Staubli VAL3: ActiviteEleve.pjx

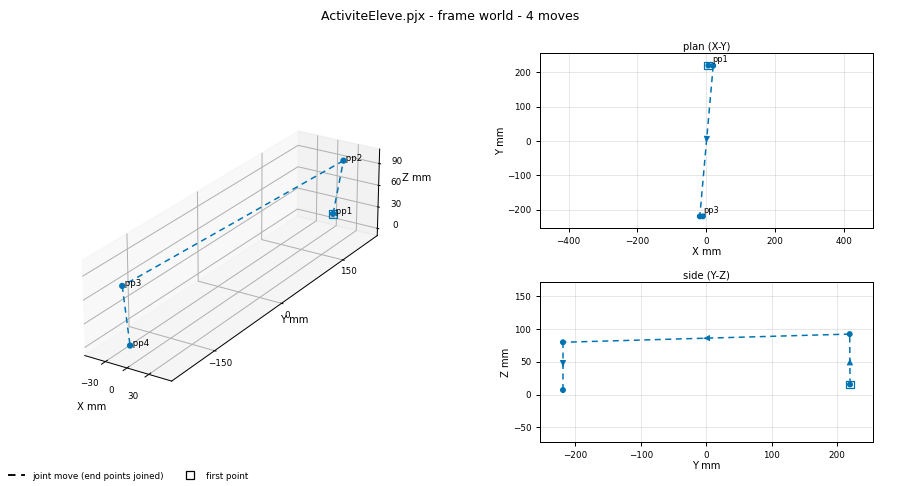
[picture p0: tool path of ActiviteEleve.pjx in frame world, 4 of 6 moves have a stored position in this frame; points joined in program order, loops and branches not executed]
--- ActiviteEleve.pjx ---
Parameters version=s7.11 stackSize=5000 millimeterUnit=true
Program file=check.pgx
Program file=comunication.pgx
Program file=coucou.pgx
Program file=jump.pgx
Program file=PickAndPlace.pgx
Program file=start.pgx
Program file=stop.pgx
Data file=ActiviteEleve.dtx
Library alias=io path=Disk://io/io.pjx

--- ActiviteEleve.dtx ---
pointRs pp1 = {x=6.500000, y=219.500000, z=15.500000, rx=-180, ry=-5.500000e-15, rz=-55.000000, fatherId=world[0]}
pointRs pp2 = {x=20.500000, y=219.000000, z=92.500000, rx=-180, ry=-5.500000e-15, rz=-55.000000, fatherId=world[0]}
pointRs pp3 = {x=-18.500000, y=-219.000000, z=80.000000, rx=180, ry=5.500000e-15, rz=125.500000, fatherId=world[0]}
pointRs pp4 = {x=-9.500000, y=-219.000000, z=7.000000, rx=180, ry=5.500000e-15, rz=123.000000, fatherId=world[0]}

--- start.pgx ---
program start()
begin
  // clean the screen
  userPage()
  cls()
  // create the 2 task
  taskCreate "comunication",10,comunication()
  delay(0.1)
  taskCreate "check",10,check()
end

--- check.pgx ---
program check()
begin
  while taskStatus("comunication")!=-1
    if taskStatus("comunication")>1
      // try to clear the buffer and resume
      clearBuffer(io:tcp_client)
      taskKill("comunication")
      wait(taskStatus("comunication")==-1)
      // create the task again from the beginning
      taskCreate "comunication",10,comunication()
    endIf
    delay(0)
  endWhile
end

--- comunication.pgx ---
program comunication()
  local string sChoixMode
  local string sClient
begin
  // clear the buffer
  clearBuffer(io:tcp_server)
  sClient="Connexion reussie"
  io:tcp_server=sClient

  putln("Un client est connecté")

  while(isKeyPressed(255)==false)
    // write
    sClient="Attente de consigne"
    io:tcp_server=sClient

    // read
    sChoixMode=io:tcp_server
    putln("Mode choisi: "+sChoixMode)

    switch sChoixMode
      //Mode coucou
      case "1"
        //on supprime les tâches en cours
        if taskStatus("jump") != -1
          taskKill("jump")
        endIf
        if taskStatus("pick&place") != -1
          taskKill("pick&place")
        endIf

        delay(0.5)

        putln("Lancement du mode coucou")
        taskCreate "coucou", 10, coucou()
      break
      //Mode jump
      case "2"
        if taskStatus("coucou") != -1
          taskKill("coucou")
        endIf
        if taskStatus("pick&place") != -1
          taskKill("pick&place")
        endIf

        delay(0.5)

        putln("Lancement du mode jump")
        taskCreate "jump", 10, jump()
      break
      //Mode pick & place
      case "3"
        if taskStatus("coucou") != -1
          taskKill("coucou")
        endIf
        if taskStatus("jump") != -1
          taskKill("jump")
        endIf

        delay(0.5)

        putln("Lancement du mode pick and place")
        taskCreate "pick&place", 10, PickAndPlace()
      break

      default
        putln(sChoixMode)
      break

    endSwitch
  endWhile
end

--- jump.pgx ---
program jump()
begin
  while true
    movej(jump1,flange,mNomSpeed)
    movej(jump2,flange,mNomSpeed)
    waitEndMove()
  endWhile
end

--- PickAndPlace.pgx ---
program PickAndPlace()
      while true
        movej(pp1, flange, mNomSpeed)
        movej(pp2, flange, mNomSpeed)
        movej(pp3, flange, mNomSpeed)
        movej(pp4, flange, mNomSpeed)
        waitEndMove()
      endWhile

--- stop.pgx ---
program stop()
begin
  clearBuffer(io:tcp_client)
  popUpMsg("Pending movement commands have been canceled")
  resetMotion()
end
